INTERFACE I_Adapter_AXIS_REF

PROPERTY getAxisRef : REFERENCE TO Tc2_MC2.AXIS_REF
GET
END_GET
END_PROPERTY

END_INTERFACE

(* stored: Version 1.1.0.1, ProductVersion 3.1.4024.12
   Itf I_Adapter_AXIS_REF: Id {5288e1c3-6908-424e-bd40-426005239927}
   Folder Status: Id {f0b191af-b924-4d43-9403-f5f55ff97497}
   Property getAxisRef: Id {f94b1389-08f4-45fa-ac95-ae70593e6ac6}
   Get Get: Id {e9d223ce-247c-48c5-87bd-7cca89be8e06} *)
